TYPE T_Ctrl_SIf_MOD_Ilk :
STRUCT
	///interlock retraction of cylinder
	bolRetract: BOOL;
	///interlock extend of cylinder
	bolExtend: BOOL;
END_STRUCT
END_TYPE

(* stored: Version 1.1.0.1, ProductVersion 3.1.0.18
   DUT T_Ctrl_SIf_MOD_Ilk: Id {eaf77187-66c6-43a0-bb08-275ef05aeecd} *)
